(*			
	RafalOS
	Rafał Osajda		20.11.2025		TC 4024.66
	Moduł przygotowania danych dla Okna zdarzeń we wszystkich trybach
*)
FUNCTION_BLOCK FB_MCHMIPrepareDataForScreen_03_XX EXTENDS FB_MCHMIPrepareDataForScreen IMPLEMENTS ITF_MCHMIPrepareDataForScreen
VAR
	itfMachineControlHMI	: ITF_MCHMIMachineControl_HMI_PrepScr_03_XX;
	refstData				: REFERENCE TO ST_MCHMIPrepareScreen_03_XX;
END_VAR

(*			
	RafalOS
	Rafał Osajda		19.11.2025		TC 4024.66
	Czyści danych przy zmienia ramki po poprzedniej ramce
*)
METHOD PUBLIC ClearAfterScreen : BOOL
VAR_INPUT
END_VAR
SUPER^.ClearAfterScreen ();
END_METHOD

METHOD PUBLIC LinkDataHMI_03_XX : BOOL
VAR_INPUT
	refstData				: REFERENCE TO ST_MCHMIPrepareScreen_03_XX;
END_VAR
THIS^.refstData REF= refstData;
END_METHOD

METHOD PUBLIC LinkMachineControlHMI : BOOL
VAR_INPUT
	fbMachineControlHMI	: ITF_MCHMIMachineControl_HMI_PrepScr_03_XX;
END_VAR
this^.itfMachineControlHMI := fbMachineControlHMI;
END_METHOD

(*			
	RafalOS
	Rafał Osajda		14.11.2025		TC 4024.66
	Metoda przygotowywania danych dla HMI 
	W niej odbywa się odpytywanie właściego elementu przez łącznik
*)
METHOD PUBLIC PrepareDataForHMI : BOOL
VAR_INPUT
END_VAR
SUPER^.PrepareDataForHMI ();
END_METHOD

(*			
	RafalOS
	Rafał Osajda		19.11.2025		TC 4024.66
	Przygotowanie ramki pood tamke do wyświetlenia - tylko przygotowanie a nie przygotowanie danych do wyświetlenia
*)
METHOD PUBLIC PrepareForScreen : BOOL
VAR_INPUT
END_VAR
SUPER^.PrepareForScreen ();
END_METHOD

END_FUNCTION_BLOCK

(* stored: Version 1.1.0.1
   POU FB_MCHMIPrepareDataForScreen_03_XX: Id {95c921f0-7619-08ed-01cb-7d69afa8090d}, SpecialFunc None
   Folder ITF_PDFS: Id {32f87cb6-0ca8-01c5-3266-7facaa29ebbf}
   Method ClearAfterScreen: Id {8d2973fc-2351-0cbe-1593-42f881e6546b}
   Method LinkDataHMI_03_XX: Id {048d1338-3482-0973-06a1-84dc14c33cc6}
   Method LinkMachineControlHMI: Id {1a975eca-2e93-0358-2e68-f9f356edf5d7}
   Method PrepareDataForHMI: Id {6c237485-98bb-06b6-3e0c-c2feceed06ba}
   Method PrepareForScreen: Id {b82a3edf-a408-0b33-02ea-fe740fb6ca57} *)
